(* IEC 61131-3 sources: teller/JD_Teller_LC2_V11/Class/CIV_Base (part 2) *)

    //save thispointer of call
    ( ( #s_CDIAS.p_CDIASAccesses^.p_This + ( s_CDIAS.ui_CDIASCounter * sizeof( t_OneCDIASAccess ) ) )$^DINT )^ := thisp$DINT;

    //increase cdias counter
    s_CDIAS.ui_CDIASCounter += 1;
  end_if;

END_FUNCTION //VIRTUAL GLOBAL CIV_Base::AddWr16Bit
//[#ENGLISH]
//=================================================================================================
//Function read id out of eeprom
//=================================================================================================
//[<Kennund]id of cdias module
//[>Place]place of cdias module
FUNCTION VIRTUAL GLOBAL CIV_Base::GetKennung
VAR_INPUT
  Place		: UDINT;
END_VAR
VAR_OUTPUT
  Kennung		: UDINT;
END_VAR
VAR
  sd_retval : DINT;
END_VAR

#ifdef IsTransparent_IS_AVAILABLE
  IF VaranIn.IsTransparent() THEN
    Kennung := 255;
    return;
  END_IF;
#endif

  //read one byte out of eeprom
(*	sd_retval := I2CReadOneByte	( AdressCDIAS 	:= ( Place * 16#100 )$UINT + 2
                , pData			:= ( #Kennung )$^USINT
                );

  //we only need one byte
  Kennung := Kennung and 16#FF;

  //look for an error
  if ( sd_retval <> VARANMANAGER_OK & b_EEPromError = TRUE ) then
    b_EEPromError := FALSE;
    Control := 0;
    VaranIn.SetState( sd_error := _ClassOk );
  end_if;
*)

  //look if class is already initialized
  if ( b_Initialized = FALSE ) then
    CIV_Init();
  end_if;

  //look if class is ok
  if ( Control = 0 ) then

    //read one byte of CDIAS - EEPROM
    sd_retval := ReadCDIASEEpromCIV(  us_cdias_place	:= ((( Place * 16#100 )$UINT + 2) shr 8 )$USINT
                    , us_offset			:= (( Place * 16#100 )$UINT + 2)$USINT
                    , ui_length			:= 1
                    , p_us_data			:= ( #Kennung )$^USINT
                    );

    //check for errors
    if ( sd_retval <> VARANMANAGER_OK ) then
      Kennung	:= 255;
    else
      //we only need one byte
      Kennung := Kennung and 16#FF;
    end_if;

  else
    Kennung	:= 255;
  end_if;

END_FUNCTION //VIRTUAL GLOBAL CIV_Base::GetKennung

//[#ENGLISH]
//=================================================================================================
//Function to activate single calls
//=================================================================================================
FUNCTION VIRTUAL GLOBAL CIV_Base::RtWork
VAR_INPUT
  EAX		: UDINT;
END_VAR
VAR_OUTPUT
  state		: UDINT;
END_VAR
VAR
  i				: UDINT;
  us_act_number	: USINT;
  p_one_cdias		: ^t_OneCDIASAccess;
  us_act_call		: USINT;
  us_act_call_old	: USINT;
  p_cdias			: ^HwBaseCDIAS;
  p_CdiasCallback	: ^t_CDIASCallback;
END_VAR

  //if class is ok
  if ( Control = 0 ) then

    //call update methods with defined priority (in differently order according to the place number)
    if ( us_cntPrioTasksRT > 0 ) then

      for i := 0 to us_cntPrioTasksRT - 1 do

        p_CdiasCallback := #a_CdiasCallBacks[ a_TasksRT[ i ].us_Place ];
        if ( p_CdiasCallback^.ud_Flags.3 = 1 ) then
          p_cdias := p_CdiasCallback^.ud_Thisp$^HwBaseCDIAS;

          //call class
          p_cdias^.UpdateRt( 0 );
        end_if;

      end_for;

    end_if;

    //check if we have a new class to call
    for i := 0 to 7 do

      p_CdiasCallback := #a_CdiasCallBacks[ i ];
      if ( p_CdiasCallback^.ud_Flags.1 = 1 ) then
        p_cdias := p_CdiasCallback^.ud_Thisp$^HwBaseCDIAS;

        //call class
        p_cdias^.UpdateRt( 0 );
      end_if;
    end_for;

    //if we have no handle return
    if ( s_CDIAS.us_HandleCounter = 0 ) then
      return;
    end_if;

    //set act number to invalid
    us_act_number 	:= 16#FF;
    us_act_call_old := 16#FF;

    //we must search in all handles
    for i := 0 to ( s_CDIAS.ui_CDIASCounter - 1 ) do

      //get one cdias strcture
      p_one_cdias := s_CDIAS.p_CDIASAccesses + ( sizeof( t_OneCDIASAccess ) * i );

      //look if it is in realtime
      if ( (p_one_cdias^.us_RTCY) AND VARAN_DOL_ISO = VARAN_DOL_ISO ) then

        //save handle number
        us_act_call := p_one_cdias^.us_CallNumber;

        //every call number is called one time
        if ( us_act_call <> us_act_call_old ) then
          us_act_call_old := us_act_call;
          p_CdiasClassRt$DINT := p_one_cdias^.p_This;

          p_CdiasClassRt^.UpDateRt( ( #p_one_cdias^.us_Handle - _IOSegment )$UDINT );
        end_if;

        //look if it is a single call (and is activated)
        if ( p_one_cdias^.us_Handle = Dmsingle ) then

          //reset single call
          p_one_cdias^.us_Handle := 0;
          //save handle number
          us_act_number := p_one_cdias^.us_CallNumber;

        end_if;

        //if handle number is same as call number change state of DO to single run
        if ( p_one_cdias^.us_CallNumber = us_act_number ) then
          if b_PayloadSupport then
            p_one_cdias^.b_DOIsRunning.StartRequest := true;
          else
          p_one_cdias^.p_HandleDO^.ucCtrlStat := VaranIn.SetRunStatus(VARAN_DO_SINGLE_RUN);
        end_if;

      end_if;

        if b_PayloadSupport then

          // p_one_cdias xxxxxxxxxxxxxxxxxxxxxxxxxxxxxxxxxxxxxxxxxxxxxxxxxxxxxxxxxxxxxxxxxxxxxxxxxxxxxxxxxxxxxxxxxxxxxxxx
          case p_one_cdias^.b_DOIsRunning of

            SR_STATE_ENABLE_ME :  // DO is not running and start request is set ----------------------------------------
              VaranIn.EnableDO(ud_DOHandle := p_one_cdias^.p_HandleDO$UDINT);
              p_one_cdias^.b_DOIsRunning  := SR_STATE_DISABLE_ME;

            SR_STATE_DISABLE_ME : // DO is running and start request is not set ----------------------------------------
              VaranIn.DisableDO(ud_DOHandle:= p_one_cdias^.p_HandleDO$UDINT);
              p_one_cdias^.b_DOIsRunning := SR_STATE_NOTHING;

            SR_STATE_LEAVE_ME_ENABLED : // DO is running and another start request is set ------------------------------
              p_one_cdias^.b_DOIsRunning := SR_STATE_DISABLE_ME;

          end_case;
        end_if;

      end_if;
    end_for;
  end_if;

  state:= READY;

END_FUNCTION //VIRTUAL GLOBAL CIV_Base::RtWork
//[#ENGLISH]
// ***************************************************************
//   This Function is Called by PostScan from DiasMasterPostScan
// ***************************************************************
FUNCTION VIRTUAL GLOBAL CIV_Base::CyWork
VAR_INPUT
  EAX		: UDINT;
END_VAR
VAR_OUTPUT
  state		: UDINT;
END_VAR
VAR
  i				: UDINT;
  us_act_number	: USINT;
  p_one_cdias		: ^t_OneCDIASAccess;
  us_act_call		: USINT;
  us_act_call_old	: USINT;
  p_cdias			: ^HwBaseCDIAS;
  p_CdiasCallback	: ^t_CDIASCallback;
END_VAR

  //if class is ok
  if ( Control = 0 ) then

    //first check if we have a new class to call
    for i := 0 to 7 do

      p_CdiasCallback	:= #a_CdiasCallBacks[ i ];

      if ( p_CdiasCallback^.ud_Flags.2 = 1 ) then
        p_cdias := p_CdiasCallback^.ud_Thisp$^HwBaseCDIAS;

        //call class
        p_cdias^.UpdataCy( 0 );
      end_if;
    end_for;

    //if we have no handle return
    if ( s_CDIAS.us_HandleCounter = 0 ) then
      return;
    end_if;

    //set act number to invalid
    us_act_number 	:= 16#FF;
    us_act_call_old	:= 16#FF;

    //we must search in all handles
    for i := 0 to ( s_CDIAS.ui_CDIASCounter - 1 ) do

      //get one cdias strcture
      p_one_cdias := s_CDIAS.p_CDIASAccesses + ( sizeof( t_OneCDIASAccess ) * i );

      //look if it is in cyclic
      if ( p_one_cdias^.us_RTCY = VARAN_DOL_ASY ) then

        //save handle number
        us_act_call := p_one_cdias^.us_CallNumber;

        //every call number is called one time
        if ( us_act_call <> us_act_call_old ) then
          us_act_call_old := us_act_call;
          p_CdiasClassCy$DINT := p_one_cdias^.p_This;

          p_CdiasClassCy^.UpDataCy( ( #p_one_cdias^.us_Handle - _IOSegment )$UDINT );
        end_if;

        //look if it is a single call (and is activated)
        if ( p_one_cdias^.us_Handle = Dmsingle) then

          //reset single call
          p_one_cdias^.us_Handle := 0;
          //save handle number
          us_act_number := p_one_cdias^.us_CallNumber;

        end_if;

        //if handle number is same as call number change state of DO to single run
        if ( p_one_cdias^.us_CallNumber = us_act_number ) then
          if b_PayloadSupport then
            p_one_cdias^.b_DOIsRunning.StartRequest := true;
          else
          p_one_cdias^.p_HandleDO^.ucCtrlStat := VaranIn.SetRunStatus(VARAN_DO_SINGLE_RUN);
          end_if;
        end_if;

        if b_PayloadSupport then

          // p_one_cdias xxxxxxxxxxxxxxxxxxxxxxxxxxxxxxxxxxxxxxxxxxxxxxxxxxxxxxxxxxxxxxxxxxxxxxxxxxxxxxxxxxxxxxxxxxxxxxxx
          case p_one_cdias^.b_DOIsRunning of

            SR_STATE_ENABLE_ME :  // DO is not running and start request is set ----------------------------------------
              VaranIn.EnableDO(ud_DOHandle := p_one_cdias^.p_HandleDO$UDINT);
              p_one_cdias^.b_DOIsRunning  := SR_STATE_DISABLE_ME;

            SR_STATE_DISABLE_ME : // DO is running and start request is not set ----------------------------------------
              VaranIn.DisableDO(ud_DOHandle:= p_one_cdias^.p_HandleDO$UDINT);
              p_one_cdias^.b_DOIsRunning := SR_STATE_NOTHING;

            SR_STATE_LEAVE_ME_ENABLED : // DO is running and another start request is set ------------------------------
              p_one_cdias^.b_DOIsRunning := SR_STATE_DISABLE_ME;

          end_case;
      end_if;

      end_if;
    end_for;
  end_if;

  state:= READY;

END_FUNCTION //VIRTUAL GLOBAL CIV_Base::CyWork
//[#ENGLISH]
//=================================================================================================
//Function to get Pll time of master
//=================================================================================================
FUNCTION VIRTUAL GLOBAL CIV_Base::GetPllTime
VAR_OUTPUT
  PllTime		: DINT;
END_VAR

  PllTime := ( VaranIn.VaranIn.GetVaranTime() / 1000000 )$DINT;

END_FUNCTION //VIRTUAL GLOBAL CIV_Base::GetPllTime
//[#ENGLISH]
//=================================================================================================
//Function to set memory error an set master off
//=================================================================================================
FUNCTION  CIV_Base::Error_ToManyCDIASAccesses

  if ( Control = 0 ) then
    Control := _MemoryFault;
    TRACE( "CIV_Base: To many CDIAS Accesses for CIV module!" );
    VaranIn.SetState( sd_error := _MemoryFault );
    VaranIn.VaranIn.SetManagerOff( e_error := Control$t_e_VaranErrors );
  end_if;

END_FUNCTION // CIV_Base::Error_ToManyCDIASAccesses
//[#ENGLISH]
//=================================================================================================
//Function to read a CDIAS - EEprom over varan bus
//=================================================================================================
//[>us_cdias_place]Place of cdias module
//[>us_offset]offset in eeprom
//[>ui_length]length of data
//[>p_us_data]pointer to data
FUNCTION  CIV_Base::ReadCDIASEEPromCIV
VAR_INPUT
  us_cdias_place		: USINT;
  us_offset			: USINT;
  ui_length			: UINT;
  p_us_data			: ^USINT;
END_VAR
VAR_OUTPUT
  sd_retval			: DINT;
END_VAR

  //init EEProm
  sd_retval := VARANTOCDIAS_iInitI2C	( uiMaster	:= ud_VaranManagerNr
                    , pucNode	:= p_NodeString
                    );

  if ( sd_retval <> VARANMANAGER_OK ) then
    return;
  end_if;

  //call OS - function to get eeprom data
  sd_retval := VARANTOCDIAS_iReadI2C( uiMaster  := ud_VaranManagerNr
                                    , pucNode   := p_NodeString
                                    , uiStation := us_cdias_place
                                    , uiOffset  := us_offset
                                    , uiLen     := ui_length
                                    , pucData   := p_us_data
                                  );

  if ( sd_retval <> VARANMANAGER_OK ) then
    return;
  end_if;

  sd_retval := VARANTOCDIAS_iExitI2C	( uiMaster	:= ud_VaranManagerNr
                    , pucNode	:= p_NodeString
                    );

END_FUNCTION // CIV_Base::ReadCDIASEEPromCIV
//[#ENGLISH]
//=================================================================================================
//Function to get retry timeout for cdias access
//=================================================================================================
//[>ud_bytes]number of bytes
//[<ud_timeout]timeout for data object
FUNCTION  CIV_Base::GetRetryTimeout
VAR_INPUT
  ud_bytes		: UDINT;
END_VAR
VAR_OUTPUT
  ud_timeout		: UDINT;
END_VAR

  //look if class is already initialized
  if ( b_Initialized = FALSE ) then
    CIV_Init();
  end_if;

  //Already got response time?
  if ud_ResponseTimeMax = 0 then
    if p_NodeInfo then
      ud_ResponseTimeMax := p_NodeInfo^.uiResponseTimeMax;
      else  // Case is possible because CIV_Init(); may fail. For example if the civ has no power supply
        ud_timeout := 0;  // Return value must be checked for 0!
        return;
    end_if;

  end_if;

  //check if Initialized is well done, else call init (cause otherwise pointer could be invalid)
  ud_timeout := ud_ResponseTimeMax + ud_bytes * VM_TIMEOUT_ONE_BYTE + ud_bytes * VM_TIMEOUT_ONE_CDIAS + VM_RETRY_TIMEOUT_STD_OFFSET;

END_FUNCTION // CIV_Base::GetRetryTimeout

FUNCTION VIRTUAL GLOBAL CIV_Base::AddCall2List
  VAR_INPUT
    Mode 	: UINT;
    RTCY 	: DINT;
    thisp 	: ^void;
    callOptions 	: USINT;
  END_VAR
  VAR_OUTPUT
    Handle 	: DINT;
  END_VAR

  //look if class is already initialized
  if ( b_Initialized = FALSE ) then
    CIV_Init();
  end_if;

  //look if CDIAS list is full
  if ( s_CDIAS.ui_CDIASCounter = s_CDIAS.ui_MaxCDIAS ) then

    Error_ToManyCDIASAccesses();
  end_if;

  //increas CDIAS counter to get right list position
  s_CDIAS.us_HandleCounter += 1;

  //look if we have realtime or cyclic
  if ( RTCY = 0 ) then
    RTCY := VARAN_DOL_ASY;
  else
    RTCY := 0;
    IF callOptions AND CALL_OPTION_RT_PRESCAN THEN
      RTCY := VARAN_DOL_ISO;
    END_IF;

    IF callOptions AND CALL_OPTION_RT_POSTSCAN THEN
      RTCY := RTCY OR CALL_OPTION_RT_POSTSCAN;
    END_IF;
  end_if;

  //get right pointer to handle in CDIAS list and manipulate it to be compatible
  Handle := ( #s_CDIAS.p_CDIASAccesses^.us_Handle + ( s_CDIAS.ui_CDIASCounter * sizeof( t_OneCDIASAccess ) ) - _IOSegment )$DINT;

  //save right handle counter
  ( ( #s_CDIAS.p_CDIASAccesses^.us_CallNumber + ( s_CDIAS.ui_CDIASCounter * sizeof( t_OneCDIASAccess ) ) )$^USINT )^ := s_CDIAS.us_HandleCounter;

  //set right call number to know which access belong to the same call
  ( ( #s_CDIAS.p_CDIASAccesses^.us_RtCy + ( s_CDIAS.ui_CDIASCounter * sizeof( t_OneCDIASAccess ) ) )$^USINT )^ := RTCY$USINT;

  //save thispointer of call
  ( ( #s_CDIAS.p_CDIASAccesses^.p_This + ( s_CDIAS.ui_CDIASCounter * sizeof( t_OneCDIASAccess ) ) )$^DINT )^ := thisp$DINT;

  //increase cdias counter
  s_CDIAS.ui_CDIASCounter += 1;

END_FUNCTION //VIRTUAL GLOBAL CIV_Base::AddCall2List
//[#ENGLISH]
//[>p_data]pointer to varan write data
//[>ud_address]address of do
FUNCTION VIRTUAL GLOBAL CIV_Base::SetNewDOAddressRd
VAR_INPUT
  p_data			: ^DINT;
  ud_address		: UDINT;
END_VAR
VAR
  p_addressRd		: ^t_VaranDOSettingsRd;
END_VAR

#ifdef IsTransparent_IS_AVAILABLE
  IF VaranIn.IsTransparent() THEN
    return;
  END_IF;
#endif

#ifdef VM_DEBUG_PAYLOAD
  // Payload not supported
  if b_PayloadSupport then
    // This method is not supporded with Payload support
    ((0)$^USINT)^ := 0;
  end_if;
#endif

  p_addressRd := p_data - VM_DO_OFFSET_RD;
  p_addressRd^.ud_Address := ud_address + ud_DeviceAddress;

END_FUNCTION //VIRTUAL GLOBAL CIV_Base::SetNewDOAddressRd
//[#ENGLISH]
//[>p_data]pointer to varan write data
//[>ud_address]address of do
FUNCTION VIRTUAL GLOBAL CIV_Base::SetNewDOAddressWr
VAR_INPUT
  p_data		: ^DINT;
  ud_address	: UDINT;
END_VAR
VAR
  p_addressWr		: ^t_VaranDOSettingsWr;
END_VAR

#ifdef IsTransparent_IS_AVAILABLE
  IF VaranIn.IsTransparent() THEN
    return;
  END_IF;
#endif

#ifdef VM_DEBUG_PAYLOAD
  // Payload not supported
  if b_PayloadSupport then
    // This method is not supporded with Payload support
    TRACE( "CIV_Base  Method not supported with Varan Payload support" );
    ((0)$^USINT)^ := 0;
  end_if;
#endif

  p_addressWr := p_data - VM_DO_OFFSET_WR;
  p_addressWr^.ud_Address := ud_address + ud_DeviceAddress;

END_FUNCTION //VIRTUAL GLOBAL CIV_Base::SetNewDOAddressWr
//[#ENGLISH]
//[>p_data]pointer to varan write data
//[>ud_address_read]read address of do
//[>ud_address_write]write address of do
FUNCTION VIRTUAL GLOBAL CIV_Base::SetNewDOAddressRdWr
VAR_INPUT
  p_data				: ^DINT;
  ud_address_read		: UDINT;
  ud_address_write	: UDINT;
END_VAR
VAR
  p_addressRdWr		: ^t_VaranDOSettingsRdWr;
END_VAR

#ifdef IsTransparent_IS_AVAILABLE
  IF VaranIn.IsTransparent() THEN
    return;
  END_IF;
#endif

#ifdef VM_DEBUG_PAYLOAD
  // Payload not supported
  if b_PayloadSupport then
    // This method is not supporded with Payload support
    TRACE( "CIV_Base Method not supported with Varan Payload support" );
    ((0)$^USINT)^ := 0;
  end_if;
#endif

  p_addressRdWr := p_data - VM_DO_OFFSET_RDWR;
  p_addressRdWr^.ud_AddressRd := ud_address_read + ud_DeviceAddress;
  p_addressRdWr^.ud_AddressWr := ud_address_write + ud_DeviceAddress;

END_FUNCTION //VIRTUAL GLOBAL CIV_Base::SetNewDOAddressRdWr
#pragma warning( disable: 73 )

//[#DEUTSCH]
//[>irqnr]0..IRQ I/O (IRQ PIN C3) | 1..IRQ Comunication (GP2 PIN A10)
FUNCTION VIRTUAL GLOBAL CIV_Base::AddCDiasIRQ
VAR_INPUT
  irqnr		: USINT;
  ActionPtr		: pVoid;
  thisp		: pVoid;
END_VAR
VAR_OUTPUT
  ok		: USINT;
END_VAR

  Trace( "Interupts on Varanbus are not supported !!! Configurationerror in object:");
  ok := 0; // only till os gives right value back

END_FUNCTION //VIRTUAL GLOBAL CIV_Base::AddCDiasIRQ
#pragma warning( default: 73 )

//[#ENGLISH]
//=================================================================================================
//Function to write a CDIAS - EEprom over varan bus (Offset 16#B0 - 16#FF)
//=================================================================================================
FUNCTION VIRTUAL GLOBAL CIV_Base::WriteEEData
VAR_INPUT
  Adress		: UDINT;
  pData		: ^USINT;
  ui_length	: UINT;
  ui_offset	: UINT;
END_VAR
VAR_OUTPUT
  retval		: DINT;
END_VAR

  if ( _RTOSVersion >= 16#1199 ) then
    //look if class is already initialized
    if ( b_Initialized = FALSE ) then
      CIV_Init();
    end_if;

    //look for length
    if ( ui_length + ui_offset > 16#100 ) then
      retval := -2;
      return;
    end_if;

    //look for length
    if ( ui_offset > 16#FF ) then		//(Offset restriction from 16#80 to 16#FF is in OS )
      retval := -3;
      return;
    end_if;

    //look if class is ok
    if ( Control = 0 ) then

      //get whole EEPROM data
      retval := WriteCDIASEEpromCIV	( us_cdias_place	:= Adress$USINT
                      , us_offset			:= ui_offset$USINT
                      , ui_length			:= ui_length
                      , p_us_data			:= pData
                      );

      //look for an error
      //check for errors
      if ( retval <> VARANMANAGER_OK ) then
        Control := retval;
//				b_EEPromError := TRUE;
        VaranIn.SetState( sd_error := _EEPromError );
      end_if;

    else
      retval := Control;
    end_if;
  else
    retval := -1;
  end_if;

END_FUNCTION //VIRTUAL GLOBAL CIV_Base::WriteEEData
//[#ENGLISH]
//=================================================================================================
//Function to write one Byte in CDIAS - EEprom over varan bus
//=================================================================================================
FUNCTION VIRTUAL GLOBAL CIV_Base::I2CWriteOneByte
VAR_INPUT
  AdressCDIAS		: UINT;
  pData		: ^USINT;
END_VAR
VAR_OUTPUT
  result		: DINT;
END_VAR

  if ( _RTOSVersion >= 16#1199 ) then
    //look if class is already initialized
    if ( b_Initialized = FALSE ) then
      CIV_Init();
    end_if;

    //look if class is ok
    if ( Control = 0 ) then

      //read one byte of CDIAS - EEPROM
      result := WriteCDIASEEpromCIV	( us_cdias_place	:= ( AdressCDIAS shr 8 )$USINT
                      , us_offset			:= AdressCDIAS$USINT
                      , ui_length			:= 1
                      , p_us_data			:= pData
                      );

      //check for errors
      if ( result <> VARANMANAGER_OK ) then
        Control := result;
//				b_EEPromError := TRUE;
        VaranIn.SetState( sd_error := _EEPromError );
      end_if;

    else
      result	:= Control;
    end_if;
  else
    result := -1;
  end_if;

END_FUNCTION //VIRTUAL GLOBAL CIV_Base::I2CWriteOneByte
//[#ENGLISH]
//=================================================================================================
//Function to write a CDIAS - EEprom over varan bus
//=================================================================================================
//[>us_cdias_place]Place of cdias module
//[>us_offset]offset in eeprom
//[>ui_length]length of data
//[>p_us_data]pointer to data
FUNCTION  CIV_Base::WriteCDIASEEPromCIV
VAR_INPUT
  us_cdias_place		: USINT;
  us_offset			: USINT;
  ui_length			: UINT;
  p_us_data			: ^USINT;
END_VAR
VAR_OUTPUT
  sd_retval			: DINT;
END_VAR

  if ( _RTOSVersion >= 16#1199 ) then
    //init EEProm
    sd_retval := VARANTOCDIAS_iInitI2C	( uiMaster	:= ud_VaranManagerNr
                      , pucNode	:= p_NodeString
                      );

    if ( sd_retval <> VARANMANAGER_OK ) then
      return;
    end_if;

    //call OS - function to get eeprom data
    sd_retval := VARANTOCDIAS_iWriteI2C(uiMaster  := ud_VaranManagerNr
                                      , pucNode   := p_NodeString
                                      , uiStation := us_cdias_place
                                      , uiOffset  := us_offset
                                      , uiLen     := ui_length
                                      , pucData   := p_us_data
                                    );

    if ( sd_retval <> VARANMANAGER_OK ) then
      return;
    end_if;

    sd_retval := VARANTOCDIAS_iExitI2C	( uiMaster	:= ud_VaranManagerNr
                      , pucNode	:= p_NodeString
                      );
  else
    sd_retval := -1;
  end_if;

END_FUNCTION // CIV_Base::WriteCDIASEEPromCIV

FUNCTION GLOBAL CIV_Base::GetRetryCounter
VAR_OUTPUT
  ud_retries		: UDINT;
END_VAR
VAR
  i		: UINT;
  p_DO	: ^t_VARANFrame;
  TempRetryCounter  : USINT;
END_VAR

  ud_retries := 0;

  //check if we have a handle
  if ( s_HandleDOs.ui_Number = 0 ) then
    return;
  end_if;

  //search handles for Retry
  for i := 0 to s_HandleDOs.ui_Number - 1 do
    p_DO := ( s_HandleDOs.p_Handles + i * sizeof( t_VARANFrame ) );

    // TempRetryCounter := p_DO^.pHandle^.ucRetryCounter;

    TempRetryCounter := VaranIn.GetRetryCounter(ud_DOHandle:=p_DO^.pHandle$UDINT );
    ud_retries += TempRetryCounter - p_DO^.us_OldRetryCounter;
    p_DO^.us_OldRetryCounter := TempRetryCounter;
  end_for;

END_FUNCTION //GLOBAL CIV_Base::GetRetryCounter
//[#ENGLISH]
//=================================================================================================
//Function to get pointer to node string
//=================================================================================================
//[<p_us_node]pointer to node string
FUNCTION VIRTUAL GLOBAL CIV_Base::GetPointer2NodeString
VAR_OUTPUT
  p_us_node		: ^USINT;
END_VAR

  p_us_node := VaranIn.GetPointer2NodeString();

END_FUNCTION //VIRTUAL GLOBAL CIV_Base::GetPointer2NodeString

FUNCTION VIRTUAL GLOBAL CIV_Base::GetObjectPath
  VAR_INPUT
    p_us_ObjectPath : ^USINT;
  END_VAR
  VAR_OUTPUT
    sd_retval 	    : DINT;
  END_VAR
  VAR
    p_us_VaranPos		: ^USINT;
  END_VAR

#ifdef IsTransparent_IS_AVAILABLE
  IF VaranIn.IsTransparent() THEN
    sd_retval := -4;
    return;
  END_IF;
#endif

  if ( p_us_ObjectPath <> NIL ) then

    p_us_VaranPos := VaranIn.GetPointer2ObjectPath();

    if ( p_us_VaranPos = NIL ) then

      sd_retval := -3;
      return;

    end_if;

    To_StdLib.MemCpy( dest 		:= p_us_ObjectPath
                    , source	:= p_us_VaranPos
                    , size		:= p_us_VaranPos^ + 1
                    );

    //if max length is reached
    if ( p_us_ObjectPath^ >= VARAN_MAX_DEPTH ) then

      sd_retval := -1;

    else

      //increase length
      p_us_ObjectPath^ += 1;

      //add escape-sequence for starting of Dias bus
      ( p_us_ObjectPath + p_us_ObjectPath^ )^ := HWT_ESCAPE_CDIAS;

      sd_retval := 0;

    end_if;

  else

    sd_retval := -2;

  end_if;

END_FUNCTION

FUNCTION VIRTUAL GLOBAL CIV_Base::SetTaskPriority
  VAR_INPUT
    us_place 	    : USINT;
    us_priority 	: USINT;
    ud_dol_type 	: UDINT;
  END_VAR
  VAR
    i1            : USINT;
    i2            : USINT;
  END_VAR

  //add task to task priority list to define the order of update tasks unaffected by the C-DIAS place
  if ( ud_dol_type = VARAN_DOL_ISO ) then

    //isochronous task
    if ( a_CdiasCallBacks [ us_place ].ud_Flags.1 = TRUE ) then

      a_CdiasCallBacks[ us_place ].ud_Flags.3 := TRUE;
      a_CdiasCallBacks[ us_place ].ud_Flags.1 := FALSE;

      for i1 := 0 to 7 do

        //found empty entry
        if ( a_TasksRT[ i1 ].us_Priority = 0 ) then

          a_TasksRT[ i1 ].us_Place    := us_place;
          a_TasksRT[ i1 ].us_Priority := us_priority;

          us_cntPrioTasksRT += 1;

          exit;

        //found entry with lower priority (higher value)
        elsif ( a_TasksRT[ i1 ].us_Priority > us_priority ) then

          //move actual and following elements backwards to get free element
          for i2 := us_cntPrioTasksRT - 1 to i1 do

            a_TasksRT [ i2 + 1 ] := a_TasksRT [ i2 ];

          end_for;

          a_TasksRT[ i1 ].us_Place    := us_place;
          a_TasksRT[ i1 ].us_Priority := us_priority;

          us_cntPrioTasksRT += 1;

          exit;

        end_if;

      end_for;

    end_if;

    //isochronous task
    if ( a_CdiasCallBacks [ us_place ].ud_Flags.5 = TRUE ) then

      a_CdiasCallBacks[ us_place ].ud_Flags.6 := TRUE;
      a_CdiasCallBacks[ us_place ].ud_Flags.5 := FALSE;

      for i1 := 0 to 7 do

        //found empty entry
        if ( a_TasksRTPostScan[ i1 ].us_Priority = 0 ) then

          a_TasksRTPostScan[ i1 ].us_Place    := us_place;
          a_TasksRTPostScan[ i1 ].us_Priority := us_priority;

          us_cntPrioTasksRTPostScan += 1;

          exit;

        //found entry with lower priority (higher value)
        elsif ( a_TasksRTPostScan[ i1 ].us_Priority > us_priority ) then

          //move actual and following elements backwards to get free element
          for i2 := us_cntPrioTasksRTPostScan - 1 to i1 do

            a_TasksRTPostScan [ i2 + 1 ] := a_TasksRTPostScan [ i2 ];

          end_for;

          a_TasksRTPostScan[ i1 ].us_Place    := us_place;
          a_TasksRTPostScan[ i1 ].us_Priority := us_priority;

          us_cntPrioTasksRTPostScan += 1;

          exit;

        end_if;

      end_for;

    end_if;

  else

    //asynchronous task
    if ( a_CdiasCallBacks [ us_place ].ud_Flags.2 = TRUE ) then

      a_CdiasCallBacks[ us_place ].ud_Flags.4 := TRUE;
      a_CdiasCallBacks[ us_place ].ud_Flags.2 := FALSE;

      for i1 := 0 to 7 do

        //found empty entry
        if ( a_TasksCY[ i1 ].us_Priority = 0 ) then

          a_TasksCY[ i1 ].us_Place    := us_place;
          a_TasksCY[ i1 ].us_Priority := us_priority;

          us_cntPrioTasksCY += 1;

          exit;

        //found entry with lower priority (higher value)
        elsif ( a_TasksCY[ i1 ].us_Priority > us_priority ) then

          //move actual and following elements backwards to get free element
          for i2 := us_cntPrioTasksCY - 1 to i1 do

            a_TasksCY [ i2 + 1 ] := a_TasksCY [ i2 ];

          end_for;

          a_TasksCY[ i1 ].us_Place    := us_place;
          a_TasksCY[ i1 ].us_Priority := us_priority;

          us_cntPrioTasksCY += 1;

          exit;

        end_if;

      end_for;

    end_if;

  end_if;

END_FUNCTION

FUNCTION VIRTUAL GLOBAL CIV_Base::SetObjectThisp
  VAR_INPUT
    p_us_ObjectPath 	: ^USINT;
    ud_thisp 	: UDINT;
  END_VAR
  VAR_OUTPUT
    sd_retval 	: DINT;
  END_VAR

#ifdef IsTransparent_IS_AVAILABLE
  IF VaranIn.IsTransparent() THEN
    sd_retval := -1;
    return;
  END_IF;
#endif

  sd_retval := VaranIn.SetObjectThisp( p_us_ObjectPath := p_us_ObjectPath
                                     , ud_thisp        := ud_thisp
                                     );

END_FUNCTION

FUNCTION VIRTUAL GLOBAL CIV_Base::GetObjectThisp
  VAR_INPUT
    p_us_ObjectPath 	: ^USINT;
  END_VAR
  VAR_OUTPUT
    ud_Thisp 	: UDINT;
  END_VAR

#ifdef IsTransparent_IS_AVAILABLE
  IF VaranIn.IsTransparent() THEN
    ud_Thisp := 0;
    return;
  END_IF;
#endif

  ud_Thisp := VaranIn.GetObjectThisp(p_us_ObjectPath := p_us_ObjectPath);

END_FUNCTION

FUNCTION VIRTUAL GLOBAL CIV_Base::Init

  Initcounter += 1;

  //check for required in 11th init run
  if Initcounter = 11 then
    CheckforRequiredError();
  end_if;

END_FUNCTION

//BLEERN001 start
FUNCTION VIRTUAL GLOBAL CIV_Base::UpdateRtPostScan
VAR
  i				: UDINT;
  us_act_number	: USINT;
  p_one_cdias		: ^t_OneCDIASAccess;
  us_act_call		: USINT;
  us_act_call_old	: USINT;
  p_cdias			: ^HwBaseCDIAS;
  p_CdiasCallback	: ^t_CDIASCallback;
END_VAR

  //if class is ok
  if ( Control = 0 ) then

    //call update methods with defined priority (in differently order according to the place number)
    if ( us_cntPrioTasksRTPostScan > 0 ) then

      for i := 0 to us_cntPrioTasksRTPostScan - 1 do

        p_CdiasCallback := #a_CdiasCallBacks[ a_TasksRTPostScan[ i ].us_Place ];
        if ( p_CdiasCallback^.ud_Flags.6 = 1 ) then
          p_cdias := p_CdiasCallback^.ud_Thisp$^HwBaseCDIAS;

          //call class
          p_cdias^.UpdateRtPostScan();
        end_if;

      end_for;

    end_if;

    //check if we have a new class to call
    for i := 0 to 7 do

      p_CdiasCallback := #a_CdiasCallBacks[ i ];
      if ( p_CdiasCallback^.ud_Flags.5 = 1 ) then
        p_cdias := p_CdiasCallback^.ud_Thisp$^HwBaseCDIAS;

        //call class
        p_cdias^.UpdateRtPostScan();
      end_if;
    end_for;

    //if we have no handle return
    if ( s_CDIAS.us_HandleCounter = 0 ) then
      return;
    end_if;

    //set act number to invalid
    us_act_number 	:= 16#FF;
    us_act_call_old := 16#FF;

    //we must search in all handles
    for i := 0 to ( s_CDIAS.ui_CDIASCounter - 1 ) do

      //get one cdias strcture
      p_one_cdias := s_CDIAS.p_CDIASAccesses + ( sizeof( t_OneCDIASAccess ) * i );

      //look if it is in realtime
      if ( (p_one_cdias^.us_RTCY) AND CALL_OPTION_RT_POSTSCAN = CALL_OPTION_RT_POSTSCAN ) then

        //save handle number
        us_act_call := p_one_cdias^.us_CallNumber;

        //every call number is called one time
        if ( us_act_call <> us_act_call_old ) then
          us_act_call_old := us_act_call;
          p_CdiasClassRt$DINT := p_one_cdias^.p_This;

          p_CdiasClassRt^.UpdateRtPostScan( ( #p_one_cdias^.us_Handle - _IOSegment )$UDINT );
        end_if;

        //look if it is a single call (and is activated)
        if ( p_one_cdias^.us_Handle = Dmsingle ) then

          //reset single call
          p_one_cdias^.us_Handle := 0;
          //save handle number
          us_act_number := p_one_cdias^.us_CallNumber;

        end_if;

        //if handle number is same as call number change state of DO to single run
        if ( p_one_cdias^.us_CallNumber = us_act_number ) then
          if b_PayloadSupport then
            p_one_cdias^.b_DOIsRunning.StartRequest := true;
          else
          p_one_cdias^.p_HandleDO^.ucCtrlStat := VaranIn.SetRunStatus(VARAN_DO_SINGLE_RUN);
        end_if;

      end_if;

        if b_PayloadSupport then

          // p_one_cdias xxxxxxxxxxxxxxxxxxxxxxxxxxxxxxxxxxxxxxxxxxxxxxxxxxxxxxxxxxxxxxxxxxxxxxxxxxxxxxxxxxxxxxxxxxxxxxxx
          case p_one_cdias^.b_DOIsRunning of

            SR_STATE_ENABLE_ME :  // DO is not running and start request is set ----------------------------------------
              VaranIn.EnableDO(ud_DOHandle := p_one_cdias^.p_HandleDO$UDINT);
              p_one_cdias^.b_DOIsRunning  := SR_STATE_DISABLE_ME;

            SR_STATE_DISABLE_ME : // DO is running and start request is not set ----------------------------------------
              VaranIn.DisableDO(ud_DOHandle:= p_one_cdias^.p_HandleDO$UDINT);
              p_one_cdias^.b_DOIsRunning := SR_STATE_NOTHING;

            SR_STATE_LEAVE_ME_ENABLED : // DO is running and another start request is set ------------------------------
              p_one_cdias^.b_DOIsRunning := SR_STATE_DISABLE_ME;

          end_case;
        end_if;

      end_if;
    end_for;
  end_if;

END_FUNCTION
//BLEERN001 end

FUNCTION VIRTUAL GLOBAL CIV_Base::AddRequiredObject
  VAR_INPUT
    thisp 	: ^void;
  END_VAR

#ifdef IsTransparent_IS_AVAILABLE
  IF VaranIn.IsTransparent() THEN
    return;
  END_IF;
#endif

  if b_NotfirstCall = false then

    p_RequiredObjects := To_StdLib.Malloc(size:=(8*sizeof(^void))); //max 8 CDIAS Module
    VaranIn.AllowRequiredError();

    VaranIn.Required := 1;

  end_if;

  b_NotfirstCall := true;

  if RequiredObjectCounter < 8 then
    (p_RequiredObjects + (RequiredObjectCounter * sizeof(^void)))^$^void := thisp;
    RequiredObjectCounter += 1;

  else
    TRACE( "CIV-CDIAS2DataMover: Too many required object classes added");
  end_if;

END_FUNCTION

#pragma warning(disable:137 )
FUNCTION VIRTUAL CIV_Base::CheckforRequiredError
  VAR
    i : UINT;
    thisp     : ^virtualbase;
    sz_name	  : array[ 0..255 ] of char;
    MyPara    : CmdStruct;
    MyResult  : results;
    UserActionRet    : DINT;
  END_VAR

  if RequiredObjectCounter > 0 then
    //--- init the newInst command
    MyPara.uiCmd := DM_CHECK_REQUIRED_ERROR;
    for i := 0 to (RequiredObjectCounter -1) do
      thisp := (p_RequiredObjects + (i * sizeof(^void)))^$^virtualbase;
      //--- init result for next call
      MyResult.aData[0] := 16#FF;
      MyResult.aData[1] := 16#FF;
      if (thisp^.NewInst(#MyPara, #MyResult) = ERROR) then
        //Required Error!
        if MyResult.aData[1] = CDIAS_MODULE then
          UserActionRet := VaranIn.UserAction.Write(input:= VARANMANAGER_CB_CDIAS_ERROR);
        else
          UserActionRet := 1;
        end_if;

        if UserActionRet <> 0 then
          _GetObjName( thisp, #sz_name[ 0 ] );
          if RequiredErrors = 0 then
            Trace ("Required Error triggerd by object(s):");
          end_if;
          Trace (#sz_name[ 0 ] );

          RequiredErrors +=1;
        end_if;
      end_if;

    end_for;

    if RequiredErrors > 0 then
      VaranIn.SetState(_CDIASRequiredError);
    end_if;

    To_StdLib.Free(p_RequiredObjects);
  end_if;

END_FUNCTION
#pragma warning(Default:137 )

FUNCTION VIRTUAL GLOBAL CIV_Base::AddMovDO
  VAR_INPUT
    ud_dol_type 	: UDINT;
    p_ud_handle 	: ^UDINT;
    p_ud_MovSettings 	: ^UDINT;
    ud_type 	: UDINT;
  END_VAR
  VAR_OUTPUT
    sd_retval 	: DINT;
  END_VAR

#ifdef IsTransparent_IS_AVAILABLE
  IF VaranIn.IsTransparent() THEN
    sd_retval := _NotInitialized;
    return;
  END_IF;
#endif

  //look if class is already initialized
  if ( b_Initialized = FALSE ) then
    CIV_Init();
  end_if;

#ifdef VM_DEBUG_PAYLOAD
  // Payload not supported
  if b_PayloadSupport then
    // This method is not supporded with Payload support
    ((0)$^USINT)^ := 0;
  end_if;
#endif

  //add a move DO
  sd_retval := VaranIn.VaranIn.AddMovDO(ud_dol_type     :=ud_dol_type
                                      , p_ud_handle     :=p_ud_handle
                                      , p_ud_MovSettings:=p_ud_MovSettings
                                      , ud_type         :=ud_type);

  // no retrycounter for move-command => don't save it into list

END_FUNCTION

FUNCTION GLOBAL CIV_Base::CIV_ReInit

  // next time the init is called, it will initialize again
  b_Initialized 	:= FALSE;

END_FUNCTION

FUNCTION VIRTUAL GLOBAL CIV_Base::Control::NewInst
  VAR_INPUT
    pPara 	: ^CmdStruct;
    pResult 	: ^Results;
  END_VAR
  VAR_OUTPUT
    ret_code 	: IprStates;
  END_VAR

  ret_code := READY;

  case pPara^.uiCmd of
    DM_ADD_PAYLOAD_DO :
        if ( AddPayloadDO(pPara:=pPara, pResult:=pResult) ) then
          ret_code := ERROR;
  end_if;

    DM_ADD_PAYLOAD_MOVE_DO :
        if ( AddMovePayloadDO(pPara:=pPara, pResult:=pResult) ) then
          ret_code := ERROR;
        end_if;

    DM_GET_PAYLOAD_RETRY_TIMEOUT :
        pResult^.aData[0]$UDINT := GetRetryTimeout(pPara^.aPara[0]$UDINT);
        if pResult^.aData[0]$UDINT = 0 then
          ret_code := ERROR;
        end_if;

    else
        ret_code := VaranIn.NewInst(pPara, pResult);
  end_case;

END_FUNCTION

FUNCTION VIRTUAL CIV_Base::AddPayloadDO
  VAR_INPUT
    pPara 	: ^CmdStruct;
    pResult 	: ^results;
  END_VAR
  VAR_OUTPUT
    sd_retval 	: DINT;
  END_VAR
  VAR
    pTemp         : ^t_VARANFrame;

    // For NewInst command
    _Para 	            : CmdStruct;
    s_paraAddDO   : t_VM_CMD_AddDO;
    s_paraGetPointers     : t_VM_CMD_GetDataPointers;
    s_PropertyValuePair : LSL_PROPERTY_VALUE_PAIR;
  END_VAR

  sd_retval := 0;

  if ud_HandleModule then

    // Add DO to DOL
    _Para.uiCmd := VM_CMD_ADD_DO;

    // Set the Module Handle to the CIV
    s_paraAddDO.ud_ModuleHandle                 := ud_HandleModule;

    // Copy over the relevant parameters
    s_paraAddDO.ud_Command                      := pPara^.aPara[0]$^t_DM_CMD_AddDO^.ud_Command;
    s_paraAddDO.p_ud_DoHandle                   := pPara^.aPara[0]$^t_DM_CMD_AddDO^.p_ud_DoHandle;
    s_paraAddDO.ud_b_DoRequired                 := pPara^.aPara[0]$^t_DM_CMD_AddDO^.ud_b_DoRequired;
    s_paraAddDO.ud_DolType                      := pPara^.aPara[0]$^t_DM_CMD_AddDO^.ud_DolType;
    s_paraAddDO.ud_OffsetRead                   := pPara^.aPara[0]$^t_DM_CMD_AddDO^.ud_OffsetRead;
    s_paraAddDO.ud_LengthRead                   := pPara^.aPara[0]$^t_DM_CMD_AddDO^.ud_LengthRead;
    s_paraAddDO.ud_OffsetWrite                  := pPara^.aPara[0]$^t_DM_CMD_AddDO^.ud_OffsetWrite;
    s_paraAddDO.ud_LengthWrite                  := pPara^.aPara[0]$^t_DM_CMD_AddDO^.ud_LengthWrite;
    s_paraAddDO.ud_PreScalerCounterThreshold    := pPara^.aPara[0]$^t_DM_CMD_AddDO^.ud_PreScalerCounterThreshold;
    s_paraAddDO.ud_PreScalerCounterStartValue   := pPara^.aPara[0]$^t_DM_CMD_AddDO^.ud_PreScalerCounterStartValue;
    s_paraAddDO.ud_Priority                     := pPara^.aPara[0]$^t_DM_CMD_AddDO^.ud_Priority;
    s_paraAddDO.ud_Filter                       := 0; // Not used by CDIAS
    s_paraAddDO.ud_Slices                       := 0; // Not used by CDIAS
    s_paraAddDO.ud_WritePayloadType             := pPara^.aPara[0]$^t_DM_CMD_AddDO^.ud_WritePayloadType;
//                                                := pPara^.aPara[0]$^t_DM_CMD_AddDO^.p_ud_DataAddr_read    // Not used
//                                                := pPara^.aPara[0]$^t_DM_CMD_AddDO^.p_ud_DataAddr_write  // Not used

    _Para.aPara[0]  := (#s_paraAddDO)$DINT;

    VaranIn.VaranIn.NewInst(#_Para, pResult);

    if pResult^.aData[0] <> VM_CMD_OK then
      sd_retval := pResult^.aData[0];
      return;
    end_if;

    // Get the Data Poiners
    _Para.uiCmd := VM_CMD_GET_DATA_POINTERS;

    // Set the Module Handle to the CIV
    s_paraGetPointers.ud_DoHandle    := s_paraAddDO.p_ud_DoHandle^;

    s_paraGetPointers.p_ud_ReadData  := pPara^.aPara[0]$^t_DM_CMD_AddDO^.p_ud_ReadData;
    s_paraGetPointers.p_ud_WriteData := pPara^.aPara[0]$^t_DM_CMD_AddDO^.p_ud_WriteData;

    _Para.aPara[0]  := (#s_paraGetPointers)$DINT;

    VaranIn.VaranIn.NewInst(#_Para, pResult);

    if pResult^.aData[0] <> VM_CMD_OK then
      return;
    end_if;

    // Set the retry timeout of the CDIAS DO
    s_PropertyValuePair.udPropertyId    := DO_PROP_RETRY_TIMEOUT;
    s_PropertyValuePair.udPropertyValue := GetRetryTimeout(ud_bytes := s_paraAddDO.ud_LengthRead + s_paraAddDO.ud_LengthWrite);

    // Check retry timeout value
    if s_PropertyValuePair.udPropertyValue = 0 then
      pResult^.aData[0]$DINT := sd_retval := VM_CMD_ERROR_INVALID_TIMEOUT;
      return;
    end_if;

    // Set Timeout
    _Para.aPara[0] := MULTI_VARAN_iSetDoProperties(s_paraAddDO.p_ud_DoHandle^, 1, #s_PropertyValuePair);
    if pResult^.aData[0]$DINT <> VM_CMD_OK then
      sd_retval := pResult^.aData[0]$DINT;
      return;
    end_if;

  else
    pResult^.uiLng := sizeof(DINT);
    pResult^.aData[0]$DINT := VM_CMD_ERROR_MODULE_HANDLE;
    return;
  end_if;

  //save handle in structure
  if ( s_HandleDOs.ui_Number = s_HandleDOs.ui_MaxNumber ) then
    s_HandleDOs.p_Handles$^void := To_StdLib.ReAlloc	( mptr		:= s_HandleDOs.p_Handles
                                                      , newsize	:= ( s_HandleDOs.ui_MaxNumber + 8 ) * sizeof( t_VARANFrame )
                                                      );

    //look for an error
    if ( s_HandleDOs.p_Handles = NIL ) then
      Control := _MemoryFault;
      VaranIn.SetState( sd_error := _MemoryFault );
      sd_retval := VARANMANAGER_NO_MEM; // Strictly speaking not a VM error, used to prevent possible overlaps in the error codes
      return;
    end_if;
    s_HandleDOs.ui_MaxNumber += 8;
  end_if;

  pTemp := s_HandleDOs.p_Handles + s_HandleDOs.ui_Number * sizeof( t_VARANFrame );

  pTemp^.pHandle := (s_paraAddDO.p_ud_DoHandle^)$^LSL_VARANFRAME;
  pTemp^.us_OldRetryCounter := 0;
  s_HandleDOs.ui_Number += 1;

END_FUNCTION

FUNCTION VIRTUAL CIV_Base::AddMovePayloadDO
  VAR_INPUT
    pPara 	: ^CmdStruct;
    pResult 	: ^results;
  END_VAR
  VAR_OUTPUT
    sd_retval 	: DINT;
  END_VAR
  VAR

    // For NewInst command
    _Para 	            : CmdStruct;
    s_paraAddMovDO   : t_VM_CMD_AddMovDo;

  END_VAR

  if ud_HandleModule then

    // Add Move DO to DOL
    _Para.uiCmd := VM_CMD_ADD_MOV_DO;

    // Pass on the parameters
    s_paraAddMovDO.p_ud_DoHandle                  := pPara^.aPara[0]$^t_DM_CMD_AddMovDo^.p_ud_DoHandle;
    s_paraAddMovDO.ud_b_DoRequired                := pPara^.aPara[0]$^t_DM_CMD_AddMovDo^.ud_b_DoRequired;
    s_paraAddMovDO.ud_DolType                     := pPara^.aPara[0]$^t_DM_CMD_AddMovDo^.ud_DolType;
    s_paraAddMovDO.ud_SourceReadDoHandle          := pPara^.aPara[0]$^t_DM_CMD_AddMovDo^.ud_SourceReadDoHandle;
    s_paraAddMovDO.ud_SourceReadOffset            := pPara^.aPara[0]$^t_DM_CMD_AddMovDo^.ud_SourceReadOffset;
    s_paraAddMovDO.ud_DestinationWriteDoHandle    := pPara^.aPara[0]$^t_DM_CMD_AddMovDo^.ud_DestinationWriteDoHandle;
    s_paraAddMovDO.ud_DestinationWriteOffset      := pPara^.aPara[0]$^t_DM_CMD_AddMovDo^.ud_DestinationWriteOffset;
    s_paraAddMovDO.ud_LengthMove                  := pPara^.aPara[0]$^t_DM_CMD_AddMovDo^.ud_LengthMove;
    s_paraAddMovDO.ud_PreScalerCounterThreshold   := pPara^.aPara[0]$^t_DM_CMD_AddMovDo^.ud_PreScalerCounterThreshold;
    s_paraAddMovDO.ud_PreScalerCounterStartValue  := pPara^.aPara[0]$^t_DM_CMD_AddMovDo^.ud_PreScalerCounterStartValue;
    s_paraAddMovDO.ud_Priority                    := pPara^.aPara[0]$^t_DM_CMD_AddMovDo^.ud_Priority;

    _Para.aPara[0]  := (#s_paraAddMovDO)$DINT;

    // new command, but we use the original result structure to get the result of the manager in the calling
    sd_retval := ( VaranIn.VaranIn.NewInst(#_Para, pResult) )$DINT;
  else
    pResult^.uiLng := sizeof(DINT);
    pResult^.aData[0]$DINT := sd_retval := VM_CMD_ERROR_MODULE_HANDLE;
  end_if;

END_FUNCTION

FUNCTION VIRTUAL GLOBAL CIV_Base::GetModuleInfo
  VAR_INPUT
    us_place 	: USINT;
  END_VAR
  VAR_OUTPUT
    p_ModuleInfo 	: ^t_s_ModulInfo;
  END_VAR

  p_ModuleInfo := NIL;

  if us_place <= 7 then
    p_ModuleInfo := #s_ModuleInfo[us_place];
    // check if module is placed
    if p_ModuleInfo^.p_This = NIL then
      p_ModuleInfo := NIL;
      return;
    end_if;
    p_ModuleInfo^.Kennung := GetKennung(us_place)$UINT;
  end_if;

END_FUNCTION
